Fanuc TP program (LS listing): P004.LS

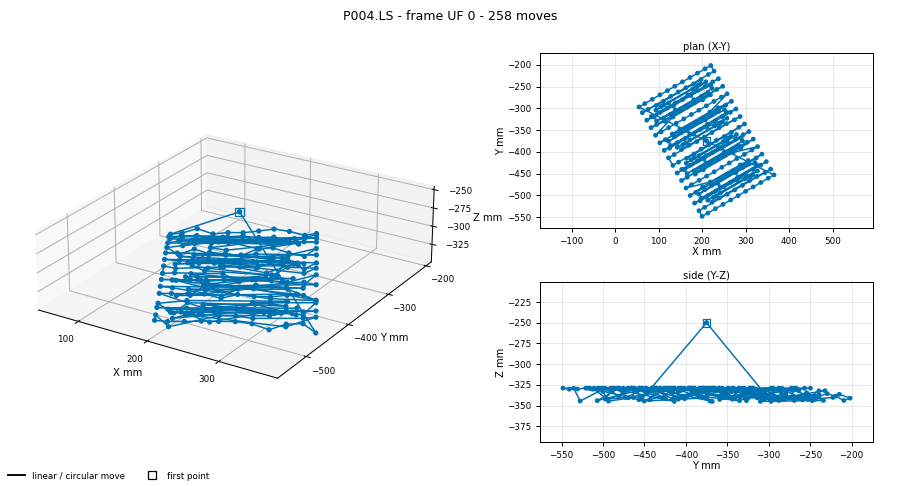
[picture p0: tool path of P004.LS in frame UF 0, 258 of 258 moves have a stored position in this frame; points joined in program order, loops and branches not executed]
/PROG  P004.LS
/ATTR
OWNER       = MNEDITOR;
COMMENT     = "";
PROG_SIZE   = 636;
CREATE      = DATE 23-01-07  TIME 11:59:14;
MODIFIED    = DATE 23-01-07  TIME 12:02:18;
FILE_NAME   = ;
VERSION     = 0;
LINE_COUNT  = 4;
MEMORY_SIZE = 992;
PROTECT     = READ_WRITE;
TCD:  STACK_SIZE	= 0,
      TASK_PRIORITY	= 50,
      TIME_SLICE	= 0,
      BUSY_LAMP_OFF	= 0,
      ABORT_REQUEST	= 0,
      PAUSE_REQUEST	= 0;
DEFAULT_GROUP	= 1,*,*,*,*;
CONTROL_CODE	= 00000000 00000000;
/MN
   1:J P[1] 100% FINE    ;
   2:L P[2] 100mm/sec CNT100    ;
   3:L P[3] 100mm/sec CNT100    ;
   4:L P[4] 100mm/sec CNT100    ;
   5:L P[5] 100mm/sec CNT100    ;
   6:L P[6] 100mm/sec CNT100    ;
   7:L P[7] 100mm/sec CNT100    ;
   8:L P[8] 100mm/sec CNT100    ;
   9:L P[9] 100mm/sec CNT100    ;
   10:L P[10] 100mm/sec CNT100    ;
   11:L P[11] 100mm/sec CNT100    ;
   12:L P[12] 100mm/sec CNT100    ;
   13:L P[13] 100mm/sec CNT100    ;
   14:L P[14] 100mm/sec CNT100    ;
   15:L P[15] 100mm/sec CNT100    ;
   16:L P[16] 100mm/sec CNT100    ;
   17:L P[17] 100mm/sec CNT100    ;
   18:L P[18] 100mm/sec CNT100    ;
   19:L P[19] 100mm/sec CNT100    ;
   20:L P[20] 100mm/sec CNT100    ;
   21:L P[21] 100mm/sec CNT100    ;
   22:L P[22] 100mm/sec CNT100    ;
   23:L P[23] 100mm/sec CNT100    ;
   24:L P[24] 100mm/sec CNT100    ;
   25:L P[25] 100mm/sec CNT100    ;
   26:L P[26] 100mm/sec CNT100    ;
   27:L P[27] 100mm/sec CNT100    ;
   28:L P[28] 100mm/sec CNT100    ;
   29:L P[29] 100mm/sec CNT100    ;
   30:L P[30] 100mm/sec CNT100    ;
   31:L P[31] 100mm/sec CNT100    ;
   32:L P[32] 100mm/sec CNT100    ;
   33:L P[33] 100mm/sec CNT100    ;
   34:L P[34] 100mm/sec CNT100    ;
   35:L P[35] 100mm/sec CNT100    ;
   36:L P[36] 100mm/sec CNT100    ;
   37:L P[37] 100mm/sec CNT100    ;
   38:L P[38] 100mm/sec CNT100    ;
   39:L P[39] 100mm/sec CNT100    ;
   40:L P[40] 100mm/sec CNT100    ;
   41:L P[41] 100mm/sec CNT100    ;
   42:L P[42] 100mm/sec CNT100    ;
   43:L P[43] 100mm/sec CNT100    ;
   44:L P[44] 100mm/sec CNT100    ;
   45:L P[45] 100mm/sec CNT100    ;
   46:L P[46] 100mm/sec CNT100    ;
   47:L P[47] 100mm/sec CNT100    ;
   48:L P[48] 100mm/sec CNT100    ;
   49:L P[49] 100mm/sec CNT100    ;
   50:L P[50] 100mm/sec CNT100    ;
   51:L P[51] 100mm/sec CNT100    ;
   52:L P[52] 100mm/sec CNT100    ;
   53:L P[53] 100mm/sec CNT100    ;
   54:L P[54] 100mm/sec CNT100    ;
   55:L P[55] 100mm/sec CNT100    ;
   56:L P[56] 100mm/sec CNT100    ;
   57:L P[57] 100mm/sec CNT100    ;
   58:L P[58] 100mm/sec CNT100    ;
   59:L P[59] 100mm/sec CNT100    ;
   60:L P[60] 100mm/sec CNT100    ;
   61:L P[61] 100mm/sec CNT100    ;
   62:L P[62] 100mm/sec CNT100    ;
   63:L P[63] 100mm/sec CNT100    ;
   64:L P[64] 100mm/sec CNT100    ;
   65:L P[65] 100mm/sec CNT100    ;
   66:L P[66] 100mm/sec CNT100    ;
   67:L P[67] 100mm/sec CNT100    ;
   68:L P[68] 100mm/sec CNT100    ;
   69:L P[69] 100mm/sec CNT100    ;
   70:L P[70] 100mm/sec CNT100    ;
   71:L P[71] 100mm/sec CNT100    ;
   72:L P[72] 100mm/sec CNT100    ;
   73:L P[73] 100mm/sec CNT100    ;
   74:L P[74] 100mm/sec CNT100    ;
   75:L P[75] 100mm/sec CNT100    ;
   76:L P[76] 100mm/sec CNT100    ;
   77:L P[77] 100mm/sec CNT100    ;
   78:L P[78] 100mm/sec CNT100    ;
   79:L P[79] 100mm/sec CNT100    ;
   80:L P[80] 100mm/sec CNT100    ;
   81:L P[81] 100mm/sec CNT100    ;
   82:L P[82] 100mm/sec CNT100    ;
   83:L P[83] 100mm/sec CNT100    ;
   84:L P[84] 100mm/sec CNT100    ;
   85:L P[85] 100mm/sec CNT100    ;
   86:L P[86] 100mm/sec CNT100    ;
   87:L P[87] 100mm/sec CNT100    ;
   88:L P[88] 100mm/sec CNT100    ;
   89:L P[89] 100mm/sec CNT100    ;
   90:L P[90] 100mm/sec CNT100    ;
   91:L P[91] 100mm/sec CNT100    ;
   92:L P[92] 100mm/sec CNT100    ;
   93:L P[93] 100mm/sec CNT100    ;
   94:L P[94] 100mm/sec CNT100    ;
   95:L P[95] 100mm/sec CNT100    ;
   96:L P[96] 100mm/sec CNT100    ;
   97:L P[97] 100mm/sec CNT100    ;
   98:L P[98] 100mm/sec CNT100    ;
   99:L P[99] 100mm/sec CNT100    ;
   100:L P[100] 100mm/sec CNT100    ;
   101:L P[101] 100mm/sec CNT100    ;
   102:L P[102] 100mm/sec CNT100    ;
   103:L P[103] 100mm/sec CNT100    ;
   104:L P[104] 100mm/sec CNT100    ;
   105:L P[105] 100mm/sec CNT100    ;
   106:L P[106] 100mm/sec CNT100    ;
   107:L P[107] 100mm/sec CNT100    ;
   108:L P[108] 100mm/sec CNT100    ;
   109:L P[109] 100mm/sec CNT100    ;
   110:L P[110] 100mm/sec CNT100    ;
   111:L P[111] 100mm/sec CNT100    ;
   112:L P[112] 100mm/sec CNT100    ;
   113:L P[113] 100mm/sec CNT100    ;
   114:L P[114] 100mm/sec CNT100    ;
   115:L P[115] 100mm/sec CNT100    ;
   116:L P[116] 100mm/sec CNT100    ;
   117:L P[117] 100mm/sec CNT100    ;
   118:L P[118] 100mm/sec CNT100    ;
   119:L P[119] 100mm/sec CNT100    ;
   120:L P[120] 100mm/sec CNT100    ;
   121:L P[121] 100mm/sec CNT100    ;
   122:L P[122] 100mm/sec CNT100    ;
   123:L P[123] 100mm/sec CNT100    ;
   124:L P[124] 100mm/sec CNT100    ;
   125:L P[125] 100mm/sec CNT100    ;
   126:L P[126] 100mm/sec CNT100    ;
   127:L P[127] 100mm/sec CNT100    ;
   128:L P[128] 100mm/sec CNT100    ;
   129:L P[129] 100mm/sec CNT100    ;
   130:L P[130] 100mm/sec CNT100    ;
   131:L P[131] 100mm/sec CNT100    ;
   132:L P[132] 100mm/sec CNT100    ;
   133:L P[133] 100mm/sec CNT100    ;
   134:L P[134] 100mm/sec CNT100    ;
   135:L P[135] 100mm/sec CNT100    ;
   136:L P[136] 100mm/sec CNT100    ;
   137:L P[137] 100mm/sec CNT100    ;
   138:L P[138] 100mm/sec CNT100    ;
   139:L P[139] 100mm/sec CNT100    ;
   140:L P[140] 100mm/sec CNT100    ;
   141:L P[141] 100mm/sec CNT100    ;
   142:L P[142] 100mm/sec CNT100    ;
   143:L P[143] 100mm/sec CNT100    ;
   144:L P[144] 100mm/sec CNT100    ;
   145:L P[145] 100mm/sec CNT100    ;
   146:L P[146] 100mm/sec CNT100    ;
   147:L P[147] 100mm/sec CNT100    ;
   148:L P[148] 100mm/sec CNT100    ;
   149:L P[149] 100mm/sec CNT100    ;
   150:L P[150] 100mm/sec CNT100    ;
   151:L P[151] 100mm/sec CNT100    ;
   152:L P[152] 100mm/sec CNT100    ;
   153:L P[153] 100mm/sec CNT100    ;
   154:L P[154] 100mm/sec CNT100    ;
   155:L P[155] 100mm/sec CNT100    ;
   156:L P[156] 100mm/sec CNT100    ;
   157:L P[157] 100mm/sec CNT100    ;
   158:L P[158] 100mm/sec CNT100    ;
   159:L P[159] 100mm/sec CNT100    ;
   160:L P[160] 100mm/sec CNT100    ;
   161:L P[161] 100mm/sec CNT100    ;
   162:L P[162] 100mm/sec CNT100    ;
   163:L P[163] 100mm/sec CNT100    ;
   164:L P[164] 100mm/sec CNT100    ;
   165:L P[165] 100mm/sec CNT100    ;
   166:L P[166] 100mm/sec CNT100    ;
   167:L P[167] 100mm/sec CNT100    ;
   168:L P[168] 100mm/sec CNT100    ;
   169:L P[169] 100mm/sec CNT100    ;
   170:L P[170] 100mm/sec CNT100    ;
   171:L P[171] 100mm/sec CNT100    ;
   172:L P[172] 100mm/sec CNT100    ;
   173:L P[173] 100mm/sec CNT100    ;
   174:L P[174] 100mm/sec CNT100    ;
   175:L P[175] 100mm/sec CNT100    ;
   176:L P[176] 100mm/sec CNT100    ;
   177:L P[177] 100mm/sec CNT100    ;
   178:L P[178] 100mm/sec CNT100    ;
   179:L P[179] 100mm/sec CNT100    ;
   180:L P[180] 100mm/sec CNT100    ;
   181:L P[181] 100mm/sec CNT100    ;
   182:L P[182] 100mm/sec CNT100    ;
   183:L P[183] 100mm/sec CNT100    ;
   184:L P[184] 100mm/sec CNT100    ;
   185:L P[185] 100mm/sec CNT100    ;
   186:L P[186] 100mm/sec CNT100    ;
   187:L P[187] 100mm/sec CNT100    ;
   188:L P[188] 100mm/sec CNT100    ;
   189:L P[189] 100mm/sec CNT100    ;
   190:L P[190] 100mm/sec CNT100    ;
   191:L P[191] 100mm/sec CNT100    ;
   192:L P[192] 100mm/sec CNT100    ;
   193:L P[193] 100mm/sec CNT100    ;
   194:L P[194] 100mm/sec CNT100    ;
   195:L P[195] 100mm/sec CNT100    ;
   196:L P[196] 100mm/sec CNT100    ;
   197:L P[197] 100mm/sec CNT100    ;
   198:L P[198] 100mm/sec CNT100    ;
   199:L P[199] 100mm/sec CNT100    ;
   200:L P[200] 100mm/sec CNT100    ;
   201:L P[201] 100mm/sec CNT100    ;
   202:L P[202] 100mm/sec CNT100    ;
   203:L P[203] 100mm/sec CNT100    ;
   204:L P[204] 100mm/sec CNT100    ;
   205:L P[205] 100mm/sec CNT100    ;
   206:L P[206] 100mm/sec CNT100    ;
   207:L P[207] 100mm/sec CNT100    ;
   208:L P[208] 100mm/sec CNT100    ;
   209:L P[209] 100mm/sec CNT100    ;
   210:L P[210] 100mm/sec CNT100    ;
   211:L P[211] 100mm/sec CNT100    ;
   212:L P[212] 100mm/sec CNT100    ;
   213:L P[213] 100mm/sec CNT100    ;
   214:L P[214] 100mm/sec CNT100    ;
   215:L P[215] 100mm/sec CNT100    ;
   216:L P[216] 100mm/sec CNT100    ;
   217:L P[217] 100mm/sec CNT100    ;
   218:L P[218] 100mm/sec CNT100    ;
   219:L P[219] 100mm/sec CNT100    ;
   220:L P[220] 100mm/sec CNT100    ;
   221:L P[221] 100mm/sec CNT100    ;
   222:L P[222] 100mm/sec CNT100    ;
   223:L P[223] 100mm/sec CNT100    ;
   224:L P[224] 100mm/sec CNT100    ;
   225:L P[225] 100mm/sec CNT100    ;
   226:L P[226] 100mm/sec CNT100    ;
   227:L P[227] 100mm/sec CNT100    ;
   228:L P[228] 100mm/sec CNT100    ;
   229:L P[229] 100mm/sec CNT100    ;
   230:L P[230] 100mm/sec CNT100    ;
   231:L P[231] 100mm/sec CNT100    ;
   232:L P[232] 100mm/sec CNT100    ;
   233:L P[233] 100mm/sec CNT100    ;
   234:L P[234] 100mm/sec CNT100    ;
   235:L P[235] 100mm/sec CNT100    ;
   236:L P[236] 100mm/sec CNT100    ;
   237:L P[237] 100mm/sec CNT100    ;
   238:L P[238] 100mm/sec CNT100    ;
   239:L P[239] 100mm/sec CNT100    ;
   240:L P[240] 100mm/sec CNT100    ;
   241:L P[241] 100mm/sec CNT100    ;
   242:L P[242] 100mm/sec CNT100    ;
   243:L P[243] 100mm/sec CNT100    ;
   244:L P[244] 100mm/sec CNT100    ;
   245:L P[245] 100mm/sec CNT100    ;
   246:L P[246] 100mm/sec CNT100    ;
   247:L P[247] 100mm/sec CNT100    ;
   248:L P[248] 100mm/sec CNT100    ;
   249:L P[249] 100mm/sec CNT100    ;
   250:L P[250] 100mm/sec CNT100    ;
   251:L P[251] 100mm/sec CNT100    ;
   252:L P[252] 100mm/sec CNT100    ;
   253:L P[253] 100mm/sec CNT100    ;
   254:L P[254] 100mm/sec CNT100    ;
   255:L P[255] 100mm/sec CNT100    ;
   256:L P[256] 100mm/sec CNT100    ;
   257:L P[257] 100mm/sec CNT100    ;
   258:L P[258] 100mm/sec CNT100    ;
/POS
P[1]{
   GP1:
	UF : 0, UT : 6,		CONFIG : 'N U T, 0, 0, 0',
	X =  210.000  mm,	Y =   -375.000  mm,	Z =   -250.000  mm,
	W =  90.000 deg,	P =   0.000 deg,	R =   90.000 deg
};
P[2]{
   GP1:
	UF : 0, UT : 6,		CONFIG : 'N U T, 0, 0, 0',
	X =  54.964  mm,	Y =   -297.033  mm,	Z =   -344.959  mm,
	W =  90.000 deg,	P =   0.000 deg,	R =   90.000 deg
};
P[3]{
   GP1:
	UF : 0, UT : 6,		CONFIG : 'N U T, 0, 0, 0',
	X =  68.285  mm,	Y =   -289.346  mm,	Z =   -342.995  mm,
	W =  90.000 deg,	P =   0.000 deg,	R =   90.000 deg
};
P[4]{
   GP1:
	UF : 0, UT : 6,		CONFIG : 'N U T, 0, 0, 0',
	X =  85.422  mm,	Y =   -279.446  mm,	Z =   -336.480  mm,
	W =  90.000 deg,	P =   0.000 deg,	R =   90.000 deg
};
P[5]{
   GP1:
	UF : 0, UT : 6,		CONFIG : 'N U T, 0, 0, 0',
	X =  102.971  mm,	Y =   -269.165  mm,	Z =   -343.776  mm,
	W =  90.000 deg,	P =   0.000 deg,	R =   90.000 deg
};
P[6]{
   GP1:
	UF : 0, UT : 6,		CONFIG : 'N U T, 0, 0, 0',
	X =  120.213  mm,	Y =   -259.452  mm,	Z =   -341.399  mm,
	W =  90.000 deg,	P =   0.000 deg,	R =   90.000 deg
};
P[7]{
   GP1:
	UF : 0, UT : 6,		CONFIG : 'N U T, 0, 0, 0',
	X =  137.188  mm,	Y =   -249.482  mm,	Z =   -341.375  mm,
	W =  90.000 deg,	P =   0.000 deg,	R =   90.000 deg
};
P[8]{
   GP1:
	UF : 0, UT : 6,		CONFIG : 'N U T, 0, 0, 0',
	X =  154.646  mm,	Y =   -239.297  mm,	Z =   -338.755  mm,
	W =  90.000 deg,	P =   0.000 deg,	R =   90.000 deg
};
P[9]{
   GP1:
	UF : 0, UT : 6,		CONFIG : 'N U T, 0, 0, 0',
	X =  171.892  mm,	Y =   -229.380  mm,	Z =   -335.633  mm,
	W =  90.000 deg,	P =   0.000 deg,	R =   90.000 deg
};
P[10]{
   GP1:
	UF : 0, UT : 6,		CONFIG : 'N U T, 0, 0, 0',
	X =  189.287  mm,	Y =   -219.340  mm,	Z =   -338.627  mm,
	W =  90.000 deg,	P =   0.000 deg,	R =   90.000 deg
};
P[11]{
   GP1:
	UF : 0, UT : 6,		CONFIG : 'N U T, 0, 0, 0',
	X =  206.728  mm,	Y =   -209.278  mm,	Z =   -343.825  mm,
	W =  90.000 deg,	P =   0.000 deg,	R =   90.000 deg
};
P[12]{
   GP1:
	UF : 0, UT : 6,		CONFIG : 'N U T, 0, 0, 0',
	X =  219.749  mm,	Y =   -201.819  mm,	Z =   -341.046  mm,
	W =  90.000 deg,	P =   0.000 deg,	R =   90.000 deg
};
P[13]{
   GP1:
	UF : 0, UT : 6,		CONFIG : 'N U T, 0, 0, 0',
	X =  227.367  mm,	Y =   -214.813  mm,	Z =   -336.366  mm,
	W =  90.000 deg,	P =   0.000 deg,	R =   90.000 deg
};
P[14]{
   GP1:
	UF : 0, UT : 6,		CONFIG : 'N U T, 0, 0, 0',
	X =  214.200  mm,	Y =   -222.393  mm,	Z =   -340.213  mm,
	W =  90.000 deg,	P =   0.000 deg,	R =   90.000 deg
};
P[15]{
   GP1:
	UF : 0, UT : 6,		CONFIG : 'N U T, 0, 0, 0',
	X =  162.666  mm,	Y =   -252.574  mm,	Z =   -342.497  mm,
	W =  90.000 deg,	P =   0.000 deg,	R =   90.000 deg
};
P[16]{
   GP1:
	UF : 0, UT : 6,		CONFIG : 'N U T, 0, 0, 0',
	X =  145.074  mm,	Y =   -262.464  mm,	Z =   -339.220  mm,
	W =  90.000 deg,	P =   0.000 deg,	R =   90.000 deg
};
P[17]{
   GP1:
	UF : 0, UT : 6,		CONFIG : 'N U T, 0, 0, 0',
	X =  127.630  mm,	Y =   -272.610  mm,	Z =   -341.020  mm,
	W =  90.000 deg,	P =   0.000 deg,	R =   90.000 deg
};
P[18]{
   GP1:
	UF : 0, UT : 6,		CONFIG : 'N U T, 0, 0, 0',
	X =  75.778  mm,	Y =   -302.469  mm,	Z =   -340.162  mm,
	W =  90.000 deg,	P =   0.000 deg,	R =   90.000 deg
};
P[19]{
   GP1:
	UF : 0, UT : 6,		CONFIG : 'N U T, 0, 0, 0',
	X =  62.714  mm,	Y =   -310.004  mm,	Z =   -344.947  mm,
	W =  90.000 deg,	P =   0.000 deg,	R =   90.000 deg
};
P[20]{
   GP1:
	UF : 0, UT : 6,		CONFIG : 'N U T, 0, 0, 0',
	X =  197.352  mm,	Y =   -233.917  mm,	Z =   -343.862  mm,
	W =  90.000 deg,	P =   0.000 deg,	R =   90.000 deg
};
P[21]{
   GP1:
	UF : 0, UT : 6,		CONFIG : 'N U T, 0, 0, 0',
	X =  180.545  mm,	Y =   -243.933  mm,	Z =   -339.685  mm,
	W =  90.000 deg,	P =   0.000 deg,	R =   90.000 deg
};
P[22]{
   GP1:
	UF : 0, UT : 6,		CONFIG : 'N U T, 0, 0, 0',
	X =  111.090  mm,	Y =   -283.819  mm,	Z =   -342.744  mm,
	W =  90.000 deg,	P =   0.000 deg,	R =   90.000 deg
};
P[23]{
   GP1:
	UF : 0, UT : 6,		CONFIG : 'N U T, 0, 0, 0',
	X =  94.177  mm,	Y =   -293.763  mm,	Z =   -339.131  mm,
	W =  90.000 deg,	P =   0.000 deg,	R =   90.000 deg
};
P[24]{
   GP1:
	UF : 0, UT : 6,		CONFIG : 'N U T, 0, 0, 0',
	X =  111.350  mm,	Y =   -292.520  mm,	Z =   -339.082  mm,
	W =  90.000 deg,	P =   0.000 deg,	R =   90.000 deg
};
P[25]{
   GP1:
	UF : 0, UT : 6,		CONFIG : 'N U T, 0, 0, 0',
	X =  189.919  mm,	Y =   -247.353  mm,	Z =   -344.029  mm,
	W =  90.000 deg,	P =   0.000 deg,	R =   90.000 deg
};
P[26]{
   GP1:
	UF : 0, UT : 6,		CONFIG : 'N U T, 0, 0, 0',
	X =  195.690  mm,	Y =   -243.952  mm,	Z =   -342.415  mm,
	W =  90.000 deg,	P =   0.000 deg,	R =   90.000 deg
};
P[27]{
   GP1:
	UF : 0, UT : 6,		CONFIG : 'N U T, 0, 0, 0',
	X =  105.186  mm,	Y =   -296.580  mm,	Z =   -339.098  mm,
	W =  90.000 deg,	P =   0.000 deg,	R =   90.000 deg
};
P[28]{
   GP1:
	UF : 0, UT : 6,		CONFIG : 'N U T, 0, 0, 0',
	X =  93.781  mm,	Y =   -304.552  mm,	Z =   -341.716  mm,
	W =  90.000 deg,	P =   0.000 deg,	R =   90.000 deg
};
P[29]{
   GP1:
	UF : 0, UT : 6,		CONFIG : 'N U T, 0, 0, 0',
	X =  122.872  mm,	Y =   -287.580  mm,	Z =   -343.772  mm,
	W =  90.000 deg,	P =   0.000 deg,	R =   90.000 deg
};
P[30]{
   GP1:
	UF : 0, UT : 6,		CONFIG : 'N U T, 0, 0, 0',
	X =  179.007  mm,	Y =   -255.068  mm,	Z =   -339.045  mm,
	W =  90.000 deg,	P =   0.000 deg,	R =   90.000 deg
};
P[31]{
   GP1:
	UF : 0, UT : 6,		CONFIG : 'N U T, 0, 0, 0',
	X =  208.523  mm,	Y =   -239.211  mm,	Z =   -336.820  mm,
	W =  90.000 deg,	P =   0.000 deg,	R =   90.000 deg
};
P[32]{
   GP1:
	UF : 0, UT : 6,		CONFIG : 'N U T, 0, 0, 0',
	X =  167.291  mm,	Y =   -269.037  mm,	Z =   -339.151  mm,
	W =  90.000 deg,	P =   0.000 deg,	R =   90.000 deg
};
P[33]{
   GP1:
	UF : 0, UT : 6,		CONFIG : 'N U T, 0, 0, 0',
	X =  83.192  mm,	Y =   -318.870  mm,	Z =   -338.828  mm,
	W =  90.000 deg,	P =   0.000 deg,	R =   90.000 deg
};
P[34]{
   GP1:
	UF : 0, UT : 6,		CONFIG : 'N U T, 0, 0, 0',
	X =  120.012  mm,	Y =   -299.352  mm,	Z =   -341.751  mm,
	W =  90.000 deg,	P =   0.000 deg,	R =   90.000 deg
};
P[35]{
   GP1:
	UF : 0, UT : 6,		CONFIG : 'N U T, 0, 0, 0',
	X =  138.499  mm,	Y =   -287.571  mm,	Z =   -341.326  mm,
	W =  90.000 deg,	P =   0.000 deg,	R =   90.000 deg
};
P[36]{
   GP1:
	UF : 0, UT : 6,		CONFIG : 'N U T, 0, 0, 0',
	X =  237.306  mm,	Y =   -232.133  mm,	Z =   -332.024  mm,
	W =  90.000 deg,	P =   0.000 deg,	R =   90.000 deg
};
P[37]{
   GP1:
	UF : 0, UT : 6,		CONFIG : 'N U T, 0, 0, 0',
	X =  224.219  mm,	Y =   -239.480  mm,	Z =   -332.129  mm,
	W =  90.000 deg,	P =   0.000 deg,	R =   90.000 deg
};
P[38]{
   GP1:
	UF : 0, UT : 6,		CONFIG : 'N U T, 0, 0, 0',
	X =  206.700  mm,	Y =   -249.866  mm,	Z =   -339.270  mm,
	W =  90.000 deg,	P =   0.000 deg,	R =   90.000 deg
};
P[39]{
   GP1:
	UF : 0, UT : 6,		CONFIG : 'N U T, 0, 0, 0',
	X =  189.366  mm,	Y =   -259.413  mm,	Z =   -342.963  mm,
	W =  90.000 deg,	P =   0.000 deg,	R =   90.000 deg
};
P[40]{
   GP1:
	UF : 0, UT : 6,		CONFIG : 'N U T, 0, 0, 0',
	X =  155.046  mm,	Y =   -279.655  mm,	Z =   -331.747  mm,
	W =  90.000 deg,	P =   0.000 deg,	R =   90.000 deg
};
P[41]{
   GP1:
	UF : 0, UT : 6,		CONFIG : 'N U T, 0, 0, 0',
	X =  103.386  mm,	Y =   -309.449  mm,	Z =   -331.657  mm,
	W =  90.000 deg,	P =   0.000 deg,	R =   90.000 deg
};
P[42]{
   GP1:
	UF : 0, UT : 6,		CONFIG : 'N U T, 0, 0, 0',
	X =  72.723  mm,	Y =   -327.289  mm,	Z =   -333.047  mm,
	W =  90.000 deg,	P =   0.000 deg,	R =   90.000 deg
};
P[43]{
   GP1:
	UF : 0, UT : 6,		CONFIG : 'N U T, 0, 0, 0',
	X =  89.392  mm,	Y =   -320.053  mm,	Z =   -331.771  mm,
	W =  90.000 deg,	P =   0.000 deg,	R =   90.000 deg
};
P[44]{
   GP1:
	UF : 0, UT : 6,		CONFIG : 'N U T, 0, 0, 0',
	X =  134.059  mm,	Y =   -294.533  mm,	Z =   -331.686  mm,
	W =  90.000 deg,	P =   0.000 deg,	R =   90.000 deg
};
P[45]{
   GP1:
	UF : 0, UT : 6,		CONFIG : 'N U T, 0, 0, 0',
	X =  173.844  mm,	Y =   -270.814  mm,	Z =   -331.661  mm,
	W =  90.000 deg,	P =   0.000 deg,	R =   90.000 deg
};
P[46]{
   GP1:
	UF : 0, UT : 6,		CONFIG : 'N U T, 0, 0, 0',
	X =  219.647  mm,	Y =   -247.088  mm,	Z =   -339.207  mm,
	W =  90.000 deg,	P =   0.000 deg,	R =   90.000 deg
};
P[47]{
   GP1:
	UF : 0, UT : 6,		CONFIG : 'N U T, 0, 0, 0',
	X =  222.521  mm,	Y =   -254.254  mm,	Z =   -334.411  mm,
	W =  90.000 deg,	P =   0.000 deg,	R =   90.000 deg
};
P[48]{
   GP1:
	UF : 0, UT : 6,		CONFIG : 'N U T, 0, 0, 0',
	X =  180.771  mm,	Y =   -280.254  mm,	Z =   -342.735  mm,
	W =  90.000 deg,	P =   0.000 deg,	R =   90.000 deg
};
P[49]{
   GP1:
	UF : 0, UT : 6,		CONFIG : 'N U T, 0, 0, 0',
	X =  138.343  mm,	Y =   -304.026  mm,	Z =   -331.765  mm,
	W =  90.000 deg,	P =   0.000 deg,	R =   90.000 deg
};
P[50]{
   GP1:
	UF : 0, UT : 6,		CONFIG : 'N U T, 0, 0, 0',
	X =  95.323  mm,	Y =   -328.988  mm,	Z =   -339.821  mm,
	W =  90.000 deg,	P =   0.000 deg,	R =   90.000 deg
};
P[51]{
   GP1:
	UF : 0, UT : 6,		CONFIG : 'N U T, 0, 0, 0',
	X =  111.227  mm,	Y =   -322.375  mm,	Z =   -329.019  mm,
	W =  90.000 deg,	P =   0.000 deg,	R =   90.000 deg
};
P[52]{
   GP1:
	UF : 0, UT : 6,		CONFIG : 'N U T, 0, 0, 0',
	X =  213.402  mm,	Y =   -263.460  mm,	Z =   -331.340  mm,
	W =  90.000 deg,	P =   0.000 deg,	R =   90.000 deg
};
P[53]{
   GP1:
	UF : 0, UT : 6,		CONFIG : 'N U T, 0, 0, 0',
	X =  198.127  mm,	Y =   -272.813  mm,	Z =   -329.019  mm,
	W =  90.000 deg,	P =   0.000 deg,	R =   90.000 deg
};
P[54]{
   GP1:
	UF : 0, UT : 6,		CONFIG : 'N U T, 0, 0, 0',
	X =  127.780  mm,	Y =   -313.727  mm,	Z =   -340.578  mm,
	W =  90.000 deg,	P =   0.000 deg,	R =   90.000 deg
};
P[55]{
   GP1:
	UF : 0, UT : 6,		CONFIG : 'N U T, 0, 0, 0',
	X =  147.349  mm,	Y =   -306.670  mm,	Z =   -342.340  mm,
	W =  90.000 deg,	P =   0.000 deg,	R =   90.000 deg
};
P[56]{
   GP1:
	UF : 0, UT : 6,		CONFIG : 'N U T, 0, 0, 0',
	X =  233.323  mm,	Y =   -256.738  mm,	Z =   -329.043  mm,
	W =  90.000 deg,	P =   0.000 deg,	R =   90.000 deg
};
P[57]{
   GP1:
	UF : 0, UT : 6,		CONFIG : 'N U T, 0, 0, 0',
	X =  247.216  mm,	Y =   -249.565  mm,	Z =   -329.013  mm,
	W =  90.000 deg,	P =   0.000 deg,	R =   90.000 deg
};
P[58]{
   GP1:
	UF : 0, UT : 6,		CONFIG : 'N U T, 0, 0, 0',
	X =  181.414  mm,	Y =   -287.792  mm,	Z =   -329.000  mm,
	W =  90.000 deg,	P =   0.000 deg,	R =   90.000 deg
};
P[59]{
   GP1:
	UF : 0, UT : 6,		CONFIG : 'N U T, 0, 0, 0',
	X =  165.019  mm,	Y =   -297.017  mm,	Z =   -329.000  mm,
	W =  90.000 deg,	P =   0.000 deg,	R =   90.000 deg
};
P[60]{
   GP1:
	UF : 0, UT : 6,		CONFIG : 'N U T, 0, 0, 0',
	X =  95.378  mm,	Y =   -337.105  mm,	Z =   -330.153  mm,
	W =  90.000 deg,	P =   0.000 deg,	R =   90.000 deg
};
P[61]{
   GP1:
	UF : 0, UT : 6,		CONFIG : 'N U T, 0, 0, 0',
	X =  82.634  mm,	Y =   -344.434  mm,	Z =   -333.012  mm,
	W =  90.000 deg,	P =   0.000 deg,	R =   90.000 deg
};
P[62]{
   GP1:
	UF : 0, UT : 6,		CONFIG : 'N U T, 0, 0, 0',
	X =  114.357  mm,	Y =   -329.935  mm,	Z =   -331.754  mm,
	W =  90.000 deg,	P =   0.000 deg,	R =   90.000 deg
};
P[63]{
   GP1:
	UF : 0, UT : 6,		CONFIG : 'N U T, 0, 0, 0',
	X =  219.042  mm,	Y =   -269.235  mm,	Z =   -329.007  mm,
	W =  90.000 deg,	P =   0.000 deg,	R =   90.000 deg
};
P[64]{
   GP1:
	UF : 0, UT : 6,		CONFIG : 'N U T, 0, 0, 0',
	X =  201.195  mm,	Y =   -280.412  mm,	Z =   -331.367  mm,
	W =  90.000 deg,	P =   0.000 deg,	R =   90.000 deg
};
P[65]{
   GP1:
	UF : 0, UT : 6,		CONFIG : 'N U T, 0, 0, 0',
	X =  132.787  mm,	Y =   -320.108  mm,	Z =   -329.026  mm,
	W =  90.000 deg,	P =   0.000 deg,	R =   90.000 deg
};
P[66]{
   GP1:
	UF : 0, UT : 6,		CONFIG : 'N U T, 0, 0, 0',
	X =  92.843  mm,	Y =   -361.854  mm,	Z =   -330.583  mm,
	W =  90.000 deg,	P =   0.000 deg,	R =   90.000 deg
};
P[67]{
   GP1:
	UF : 0, UT : 6,		CONFIG : 'N U T, 0, 0, 0',
	X =  105.822  mm,	Y =   -354.322  mm,	Z =   -340.290  mm,
	W =  90.000 deg,	P =   0.000 deg,	R =   90.000 deg
};
P[68]{
   GP1:
	UF : 0, UT : 6,		CONFIG : 'N U T, 0, 0, 0',
	X =  123.080  mm,	Y =   -344.334  mm,	Z =   -332.068  mm,
	W =  90.000 deg,	P =   0.000 deg,	R =   90.000 deg
};
P[69]{
   GP1:
	UF : 0, UT : 6,		CONFIG : 'N U T, 0, 0, 0',
	X =  140.433  mm,	Y =   -334.388  mm,	Z =   -338.788  mm,
	W =  90.000 deg,	P =   0.000 deg,	R =   90.000 deg
};
P[70]{
   GP1:
	UF : 0, UT : 6,		CONFIG : 'N U T, 0, 0, 0',
	X =  157.769  mm,	Y =   -324.401  mm,	Z =   -340.163  mm,
	W =  90.000 deg,	P =   0.000 deg,	R =   90.000 deg
};
P[71]{
   GP1:
	UF : 0, UT : 6,		CONFIG : 'N U T, 0, 0, 0',
	X =  175.019  mm,	Y =   -314.311  mm,	Z =   -340.185  mm,
	W =  90.000 deg,	P =   0.000 deg,	R =   90.000 deg
};
P[72]{
   GP1:
	UF : 0, UT : 6,		CONFIG : 'N U T, 0, 0, 0',
	X =  192.396  mm,	Y =   -304.462  mm,	Z =   -330.805  mm,
	W =  90.000 deg,	P =   0.000 deg,	R =   90.000 deg
};
P[73]{
   GP1:
	UF : 0, UT : 6,		CONFIG : 'N U T, 0, 0, 0',
	X =  209.657  mm,	Y =   -294.289  mm,	Z =   -329.043  mm,
	W =  90.000 deg,	P =   0.000 deg,	R =   90.000 deg
};
P[74]{
   GP1:
	UF : 0, UT : 6,		CONFIG : 'N U T, 0, 0, 0',
	X =  227.005  mm,	Y =   -284.264  mm,	Z =   -335.665  mm,
	W =  90.000 deg,	P =   0.000 deg,	R =   90.000 deg
};
P[75]{
   GP1:
	UF : 0, UT : 6,		CONFIG : 'N U T, 0, 0, 0',
	X =  244.227  mm,	Y =   -274.352  mm,	Z =   -340.182  mm,
	W =  90.000 deg,	P =   0.000 deg,	R =   90.000 deg
};
P[76]{
   GP1:
	UF : 0, UT : 6,		CONFIG : 'N U T, 0, 0, 0',
	X =  257.160  mm,	Y =   -266.755  mm,	Z =   -329.000  mm,
	W =  90.000 deg,	P =   0.000 deg,	R =   90.000 deg
};
P[77]{
   GP1:
	UF : 0, UT : 6,		CONFIG : 'N U T, 0, 0, 0',
	X =  217.457  mm,	Y =   -308.775  mm,	Z =   -336.833  mm,
	W =  90.000 deg,	P =   0.000 deg,	R =   90.000 deg
};
P[78]{
   GP1:
	UF : 0, UT : 6,		CONFIG : 'N U T, 0, 0, 0',
	X =  148.690  mm,	Y =   -348.108  mm,	Z =   -329.127  mm,
	W =  90.000 deg,	P =   0.000 deg,	R =   90.000 deg
};
P[79]{
   GP1:
	UF : 0, UT : 6,		CONFIG : 'N U T, 0, 0, 0',
	X =  131.305  mm,	Y =   -359.163  mm,	Z =   -342.666  mm,
	W =  90.000 deg,	P =   0.000 deg,	R =   90.000 deg
};
P[80]{
   GP1:
	UF : 0, UT : 6,		CONFIG : 'N U T, 0, 0, 0',
	X =  236.196  mm,	Y =   -298.720  mm,	Z =   -330.229  mm,
	W =  90.000 deg,	P =   0.000 deg,	R =   90.000 deg
};
P[81]{
   GP1:
	UF : 0, UT : 6,		CONFIG : 'N U T, 0, 0, 0',
	X =  267.157  mm,	Y =   -284.013  mm,	Z =   -329.000  mm,
	W =  90.000 deg,	P =   0.000 deg,	R =   90.000 deg
};
P[82]{
   GP1:
	UF : 0, UT : 6,		CONFIG : 'N U T, 0, 0, 0',
	X =  201.291  mm,	Y =   -321.927  mm,	Z =   -329.001  mm,
	W =  90.000 deg,	P =   0.000 deg,	R =   90.000 deg
};
P[83]{
   GP1:
	UF : 0, UT : 6,		CONFIG : 'N U T, 0, 0, 0',
	X =  185.095  mm,	Y =   -331.576  mm,	Z =   -330.542  mm,
	W =  90.000 deg,	P =   0.000 deg,	R =   90.000 deg
};
P[84]{
   GP1:
	UF : 0, UT : 6,		CONFIG : 'N U T, 0, 0, 0',
	X =  115.534  mm,	Y =   -372.015  mm,	Z =   -329.000  mm,
	W =  90.000 deg,	P =   0.000 deg,	R =   90.000 deg
};
P[85]{
   GP1:
	UF : 0, UT : 6,		CONFIG : 'N U T, 0, 0, 0',
	X =  102.734  mm,	Y =   -379.332  mm,	Z =   -329.028  mm,
	W =  90.000 deg,	P =   0.000 deg,	R =   90.000 deg
};
P[86]{
   GP1:
	UF : 0, UT : 6,		CONFIG : 'N U T, 0, 0, 0',
	X =  167.910  mm,	Y =   -342.172  mm,	Z =   -329.000  mm,
	W =  90.000 deg,	P =   0.000 deg,	R =   90.000 deg
};
P[87]{
   GP1:
	UF : 0, UT : 6,		CONFIG : 'N U T, 0, 0, 0',
	X =  254.271  mm,	Y =   -292.688  mm,	Z =   -341.050  mm,
	W =  90.000 deg,	P =   0.000 deg,	R =   90.000 deg
};
P[88]{
   GP1:
	UF : 0, UT : 6,		CONFIG : 'N U T, 0, 0, 0',
	X =  222.397  mm,	Y =   -315.138  mm,	Z =   -330.212  mm,
	W =  90.000 deg,	P =   0.000 deg,	R =   90.000 deg
};
P[89]{
   GP1:
	UF : 0, UT : 6,		CONFIG : 'N U T, 0, 0, 0',
	X =  151.725  mm,	Y =   -355.659  mm,	Z =   -329.013  mm,
	W =  90.000 deg,	P =   0.000 deg,	R =   90.000 deg
};
P[90]{
   GP1:
	UF : 0, UT : 6,		CONFIG : 'N U T, 0, 0, 0',
	X =  136.256  mm,	Y =   -365.631  mm,	Z =   -329.000  mm,
	W =  90.000 deg,	P =   0.000 deg,	R =   90.000 deg
};
P[91]{
   GP1:
	UF : 0, UT : 6,		CONFIG : 'N U T, 0, 0, 0',
	X =  238.230  mm,	Y =   -306.479  mm,	Z =   -331.261  mm,
	W =  90.000 deg,	P =   0.000 deg,	R =   90.000 deg
};
P[92]{
   GP1:
	UF : 0, UT : 6,		CONFIG : 'N U T, 0, 0, 0',
	X =  207.228  mm,	Y =   -326.792  mm,	Z =   -344.003  mm,
	W =  90.000 deg,	P =   0.000 deg,	R =   90.000 deg
};
P[93]{
   GP1:
	UF : 0, UT : 6,		CONFIG : 'N U T, 0, 0, 0',
	X =  165.371  mm,	Y =   -351.259  mm,	Z =   -335.727  mm,
	W =  90.000 deg,	P =   0.000 deg,	R =   90.000 deg
};
P[94]{
   GP1:
	UF : 0, UT : 6,		CONFIG : 'N U T, 0, 0, 0',
	X =  122.935  mm,	Y =   -375.735  mm,	Z =   -330.203  mm,
	W =  90.000 deg,	P =   0.000 deg,	R =   90.000 deg
};
P[95]{
   GP1:
	UF : 0, UT : 6,		CONFIG : 'N U T, 0, 0, 0',
	X =  251.034  mm,	Y =   -303.404  mm,	Z =   -336.716  mm,
	W =  90.000 deg,	P =   0.000 deg,	R =   90.000 deg
};
P[96]{
   GP1:
	UF : 0, UT : 6,		CONFIG : 'N U T, 0, 0, 0',
	X =  255.794  mm,	Y =   -309.411  mm,	Z =   -336.576  mm,
	W =  90.000 deg,	P =   0.000 deg,	R =   90.000 deg
};
P[97]{
   GP1:
	UF : 0, UT : 6,		CONFIG : 'N U T, 0, 0, 0',
	X =  171.631  mm,	Y =   -359.385  mm,	Z =   -339.120  mm,
	W =  90.000 deg,	P =   0.000 deg,	R =   90.000 deg
};
P[98]{
   GP1:
	UF : 0, UT : 6,		CONFIG : 'N U T, 0, 0, 0',
	X =  211.999  mm,	Y =   -337.291  mm,	Z =   -331.382  mm,
	W =  90.000 deg,	P =   0.000 deg,	R =   90.000 deg
};
P[99]{
   GP1:
	UF : 0, UT : 6,		CONFIG : 'N U T, 0, 0, 0',
	X =  127.390  mm,	Y =   -385.610  mm,	Z =   -331.661  mm,
	W =  90.000 deg,	P =   0.000 deg,	R =   90.000 deg
};
P[100]{
   GP1:
	UF : 0, UT : 6,		CONFIG : 'N U T, 0, 0, 0',
	X =  112.767  mm,	Y =   -396.676  mm,	Z =   -329.000  mm,
	W =  90.000 deg,	P =   0.000 deg,	R =   90.000 deg
};
P[101]{
   GP1:
	UF : 0, UT : 6,		CONFIG : 'N U T, 0, 0, 0',
	X =  143.369  mm,	Y =   -379.012  mm,	Z =   -329.000  mm,
	W =  90.000 deg,	P =   0.000 deg,	R =   90.000 deg
};
P[102]{
   GP1:
	UF : 0, UT : 6,		CONFIG : 'N U T, 0, 0, 0',
	X =  160.556  mm,	Y =   -369.393  mm,	Z =   -329.029  mm,
	W =  90.000 deg,	P =   0.000 deg,	R =   90.000 deg
};
P[103]{
   GP1:
	UF : 0, UT : 6,		CONFIG : 'N U T, 0, 0, 0',
	X =  194.810  mm,	Y =   -349.163  mm,	Z =   -329.000  mm,
	W =  90.000 deg,	P =   0.000 deg,	R =   90.000 deg
};
P[104]{
   GP1:
	UF : 0, UT : 6,		CONFIG : 'N U T, 0, 0, 0',
	X =  246.781  mm,	Y =   -319.004  mm,	Z =   -329.000  mm,
	W =  90.000 deg,	P =   0.000 deg,	R =   90.000 deg
};
P[105]{
   GP1:
	UF : 0, UT : 6,		CONFIG : 'N U T, 0, 0, 0',
	X =  264.592  mm,	Y =   -309.341  mm,	Z =   -339.203  mm,
	W =  90.000 deg,	P =   0.000 deg,	R =   90.000 deg
};
P[106]{
   GP1:
	UF : 0, UT : 6,		CONFIG : 'N U T, 0, 0, 0',
	X =  277.449  mm,	Y =   -301.566  mm,	Z =   -330.833  mm,
	W =  90.000 deg,	P =   0.000 deg,	R =   90.000 deg
};
P[107]{
   GP1:
	UF : 0, UT : 6,		CONFIG : 'N U T, 0, 0, 0',
	X =  230.019  mm,	Y =   -329.393  mm,	Z =   -329.028  mm,
	W =  90.000 deg,	P =   0.000 deg,	R =   90.000 deg
};
P[108]{
   GP1:
	UF : 0, UT : 6,		CONFIG : 'N U T, 0, 0, 0',
	X =  125.050  mm,	Y =   -391.579  mm,	Z =   -334.380  mm,
	W =  90.000 deg,	P =   0.000 deg,	R =   90.000 deg
};
P[109]{
   GP1:
	UF : 0, UT : 6,		CONFIG : 'N U T, 0, 0, 0',
	X =  179.919  mm,	Y =   -359.513  mm,	Z =   -329.008  mm,
	W =  90.000 deg,	P =   0.000 deg,	R =   90.000 deg
};
P[110]{
   GP1:
	UF : 0, UT : 6,		CONFIG : 'N U T, 0, 0, 0',
	X =  210.213  mm,	Y =   -343.666  mm,	Z =   -329.000  mm,
	W =  90.000 deg,	P =   0.000 deg,	R =   90.000 deg
};
P[111]{
   GP1:
	UF : 0, UT : 6,		CONFIG : 'N U T, 0, 0, 0',
	X =  256.759  mm,	Y =   -323.038  mm,	Z =   -329.000  mm,
	W =  90.000 deg,	P =   0.000 deg,	R =   90.000 deg
};
P[112]{
   GP1:
	UF : 0, UT : 6,		CONFIG : 'N U T, 0, 0, 0',
	X =  228.321  mm,	Y =   -340.634  mm,	Z =   -341.366  mm,
	W =  90.000 deg,	P =   0.000 deg,	R =   90.000 deg
};
P[113]{
   GP1:
	UF : 0, UT : 6,		CONFIG : 'N U T, 0, 0, 0',
	X =  171.874  mm,	Y =   -373.116  mm,	Z =   -329.042  mm,
	W =  90.000 deg,	P =   0.000 deg,	R =   90.000 deg
};
P[114]{
   GP1:
	UF : 0, UT : 6,		CONFIG : 'N U T, 0, 0, 0',
	X =  142.948  mm,	Y =   -389.644  mm,	Z =   -329.002  mm,
	W =  90.000 deg,	P =   0.000 deg,	R =   90.000 deg
};
P[115]{
   GP1:
	UF : 0, UT : 6,		CONFIG : 'N U T, 0, 0, 0',
	X =  155.686  mm,	Y =   -383.722  mm,	Z =   -329.013  mm,
	W =  90.000 deg,	P =   0.000 deg,	R =   90.000 deg
};
P[116]{
   GP1:
	UF : 0, UT : 6,		CONFIG : 'N U T, 0, 0, 0',
	X =  246.698  mm,	Y =   -331.373  mm,	Z =   -329.036  mm,
	W =  90.000 deg,	P =   0.000 deg,	R =   90.000 deg
};
P[117]{
   GP1:
	UF : 0, UT : 6,		CONFIG : 'N U T, 0, 0, 0',
	X =  240.343  mm,	Y =   -335.183  mm,	Z =   -344.054  mm,
	W =  90.000 deg,	P =   0.000 deg,	R =   90.000 deg
};
P[118]{
   GP1:
	UF : 0, UT : 6,		CONFIG : 'N U T, 0, 0, 0',
	X =  162.006  mm,	Y =   -380.425  mm,	Z =   -339.105  mm,
	W =  90.000 deg,	P =   0.000 deg,	R =   90.000 deg
};
P[119]{
   GP1:
	UF : 0, UT : 6,		CONFIG : 'N U T, 0, 0, 0',
	X =  152.570  mm,	Y =   -394.661  mm,	Z =   -329.000  mm,
	W =  90.000 deg,	P =   0.000 deg,	R =   90.000 deg
};
P[120]{
   GP1:
	UF : 0, UT : 6,		CONFIG : 'N U T, 0, 0, 0',
	X =  169.614  mm,	Y =   -384.897  mm,	Z =   -331.867  mm,
	W =  90.000 deg,	P =   0.000 deg,	R =   90.000 deg
};
P[121]{
   GP1:
	UF : 0, UT : 6,		CONFIG : 'N U T, 0, 0, 0',
	X =  238.902  mm,	Y =   -344.786  mm,	Z =   -340.586  mm,
	W =  90.000 deg,	P =   0.000 deg,	R =   90.000 deg
};
P[122]{
   GP1:
	UF : 0, UT : 6,		CONFIG : 'N U T, 0, 0, 0',
	X =  255.708  mm,	Y =   -335.320  mm,	Z =   -329.019  mm,
	W =  90.000 deg,	P =   0.000 deg,	R =   90.000 deg
};
P[123]{
   GP1:
	UF : 0, UT : 6,		CONFIG : 'N U T, 0, 0, 0',
	X =  287.230  mm,	Y =   -318.953  mm,	Z =   -329.000  mm,
	W =  90.000 deg,	P =   0.000 deg,	R =   90.000 deg
};
P[124]{
   GP1:
	UF : 0, UT : 6,		CONFIG : 'N U T, 0, 0, 0',
	X =  274.144  mm,	Y =   -326.412  mm,	Z =   -336.348  mm,
	W =  90.000 deg,	P =   0.000 deg,	R =   90.000 deg
};
P[125]{
   GP1:
	UF : 0, UT : 6,		CONFIG : 'N U T, 0, 0, 0',
	X =  222.566  mm,	Y =   -355.680  mm,	Z =   -330.140  mm,
	W =  90.000 deg,	P =   0.000 deg,	R =   90.000 deg
};
P[126]{
   GP1:
	UF : 0, UT : 6,		CONFIG : 'N U T, 0, 0, 0',
	X =  205.127  mm,	Y =   -366.356  mm,	Z =   -329.002  mm,
	W =  90.000 deg,	P =   0.000 deg,	R =   90.000 deg
};
P[127]{
   GP1:
	UF : 0, UT : 6,		CONFIG : 'N U T, 0, 0, 0',
	X =  187.649  mm,	Y =   -376.444  mm,	Z =   -329.038  mm,
	W =  90.000 deg,	P =   0.000 deg,	R =   90.000 deg
};
P[128]{
   GP1:
	UF : 0, UT : 6,		CONFIG : 'N U T, 0, 0, 0',
	X =  135.693  mm,	Y =   -406.364  mm,	Z =   -332.079  mm,
	W =  90.000 deg,	P =   0.000 deg,	R =   90.000 deg
};
P[129]{
   GP1:
	UF : 0, UT : 6,		CONFIG : 'N U T, 0, 0, 0',
	X =  122.715  mm,	Y =   -413.804  mm,	Z =   -329.001  mm,
	W =  90.000 deg,	P =   0.000 deg,	R =   90.000 deg
};
P[130]{
   GP1:
	UF : 0, UT : 6,		CONFIG : 'N U T, 0, 0, 0',
	X =  132.757  mm,	Y =   -431.210  mm,	Z =   -329.959  mm,
	W =  90.000 deg,	P =   0.000 deg,	R =   90.000 deg
};
P[131]{
   GP1:
	UF : 0, UT : 6,		CONFIG : 'N U T, 0, 0, 0',
	X =  145.670  mm,	Y =   -423.684  mm,	Z =   -329.000  mm,
	W =  90.000 deg,	P =   0.000 deg,	R =   90.000 deg
};
P[132]{
   GP1:
	UF : 0, UT : 6,		CONFIG : 'N U T, 0, 0, 0',
	X =  197.579  mm,	Y =   -393.900  mm,	Z =   -329.018  mm,
	W =  90.000 deg,	P =   0.000 deg,	R =   90.000 deg
};
P[133]{
   GP1:
	UF : 0, UT : 6,		CONFIG : 'N U T, 0, 0, 0',
	X =  214.967  mm,	Y =   -383.755  mm,	Z =   -339.766  mm,
	W =  90.000 deg,	P =   0.000 deg,	R =   90.000 deg
};
P[134]{
   GP1:
	UF : 0, UT : 6,		CONFIG : 'N U T, 0, 0, 0',
	X =  232.673  mm,	Y =   -373.776  mm,	Z =   -336.847  mm,
	W =  90.000 deg,	P =   0.000 deg,	R =   90.000 deg
};
P[135]{
   GP1:
	UF : 0, UT : 6,		CONFIG : 'N U T, 0, 0, 0',
	X =  284.419  mm,	Y =   -343.550  mm,	Z =   -342.364  mm,
	W =  90.000 deg,	P =   0.000 deg,	R =   90.000 deg
};
P[136]{
   GP1:
	UF : 0, UT : 6,		CONFIG : 'N U T, 0, 0, 0',
	X =  297.248  mm,	Y =   -336.060  mm,	Z =   -329.024  mm,
	W =  90.000 deg,	P =   0.000 deg,	R =   90.000 deg
};
P[137]{
   GP1:
	UF : 0, UT : 6,		CONFIG : 'N U T, 0, 0, 0',
	X =  267.211  mm,	Y =   -355.124  mm,	Z =   -338.981  mm,
	W =  90.000 deg,	P =   0.000 deg,	R =   90.000 deg
};
P[138]{
   GP1:
	UF : 0, UT : 6,		CONFIG : 'N U T, 0, 0, 0',
	X =  164.270  mm,	Y =   -414.926  mm,	Z =   -329.021  mm,
	W =  90.000 deg,	P =   0.000 deg,	R =   90.000 deg
};
P[139]{
   GP1:
	UF : 0, UT : 6,		CONFIG : 'N U T, 0, 0, 0',
	X =  181.158  mm,	Y =   -405.144  mm,	Z =   -339.099  mm,
	W =  90.000 deg,	P =   0.000 deg,	R =   90.000 deg
};
P[140]{
   GP1:
	UF : 0, UT : 6,		CONFIG : 'N U T, 0, 0, 0',
	X =  250.625  mm,	Y =   -365.135  mm,	Z =   -329.123  mm,
	W =  90.000 deg,	P =   0.000 deg,	R =   90.000 deg
};
P[141]{
   GP1:
	UF : 0, UT : 6,		CONFIG : 'N U T, 0, 0, 0',
	X =  266.312  mm,	Y =   -364.946  mm,	Z =   -332.108  mm,
	W =  90.000 deg,	P =   0.000 deg,	R =   90.000 deg
};
P[142]{
   GP1:
	UF : 0, UT : 6,		CONFIG : 'N U T, 0, 0, 0',
	X =  260.098  mm,	Y =   -368.362  mm,	Z =   -329.014  mm,
	W =  90.000 deg,	P =   0.000 deg,	R =   90.000 deg
};
P[143]{
   GP1:
	UF : 0, UT : 6,		CONFIG : 'N U T, 0, 0, 0',
	X =  181.653  mm,	Y =   -413.645  mm,	Z =   -339.826  mm,
	W =  90.000 deg,	P =   0.000 deg,	R =   90.000 deg
};
P[144]{
   GP1:
	UF : 0, UT : 6,		CONFIG : 'N U T, 0, 0, 0',
	X =  174.967  mm,	Y =   -417.987  mm,	Z =   -329.000  mm,
	W =  90.000 deg,	P =   0.000 deg,	R =   90.000 deg
};
P[145]{
   GP1:
	UF : 0, UT : 6,		CONFIG : 'N U T, 0, 0, 0',
	X =  248.912  mm,	Y =   -376.390  mm,	Z =   -329.117  mm,
	W =  90.000 deg,	P =   0.000 deg,	R =   90.000 deg
};
P[146]{
   GP1:
	UF : 0, UT : 6,		CONFIG : 'N U T, 0, 0, 0',
	X =  192.836  mm,	Y =   -408.880  mm,	Z =   -342.211  mm,
	W =  90.000 deg,	P =   0.000 deg,	R =   90.000 deg
};
P[147]{
   GP1:
	UF : 0, UT : 6,		CONFIG : 'N U T, 0, 0, 0',
	X =  163.435  mm,	Y =   -426.067  mm,	Z =   -329.045  mm,
	W =  90.000 deg,	P =   0.000 deg,	R =   90.000 deg
};
P[148]{
   GP1:
	UF : 0, UT : 6,		CONFIG : 'N U T, 0, 0, 0',
	X =  278.644  mm,	Y =   -360.412  mm,	Z =   -329.000  mm,
	W =  90.000 deg,	P =   0.000 deg,	R =   90.000 deg
};
P[149]{
   GP1:
	UF : 0, UT : 6,		CONFIG : 'N U T, 0, 0, 0',
	X =  237.200  mm,	Y =   -390.225  mm,	Z =   -329.043  mm,
	W =  90.000 deg,	P =   0.000 deg,	R =   90.000 deg
};
P[150]{
   GP1:
	UF : 0, UT : 6,		CONFIG : 'N U T, 0, 0, 0',
	X =  153.129  mm,	Y =   -440.137  mm,	Z =   -330.554  mm,
	W =  90.000 deg,	P =   0.000 deg,	R =   90.000 deg
};
P[151]{
   GP1:
	UF : 0, UT : 6,		CONFIG : 'N U T, 0, 0, 0',
	X =  259.444  mm,	Y =   -380.403  mm,	Z =   -329.000  mm,
	W =  90.000 deg,	P =   0.000 deg,	R =   90.000 deg
};
P[152]{
   GP1:
	UF : 0, UT : 6,		CONFIG : 'N U T, 0, 0, 0',
	X =  208.491  mm,	Y =   -408.857  mm,	Z =   -329.013  mm,
	W =  90.000 deg,	P =   0.000 deg,	R =   90.000 deg
};
P[153]{
   GP1:
	UF : 0, UT : 6,		CONFIG : 'N U T, 0, 0, 0',
	X =  190.036  mm,	Y =   -420.531  mm,	Z =   -329.068  mm,
	W =  90.000 deg,	P =   0.000 deg,	R =   90.000 deg
};
P[154]{
   GP1:
	UF : 0, UT : 6,		CONFIG : 'N U T, 0, 0, 0',
	X =  142.640  mm,	Y =   -448.526  mm,	Z =   -329.028  mm,
	W =  90.000 deg,	P =   0.000 deg,	R =   90.000 deg
};
P[155]{
   GP1:
	UF : 0, UT : 6,		CONFIG : 'N U T, 0, 0, 0',
	X =  173.073  mm,	Y =   -430.710  mm,	Z =   -329.000  mm,
	W =  90.000 deg,	P =   0.000 deg,	R =   90.000 deg
};
P[156]{
   GP1:
	UF : 0, UT : 6,		CONFIG : 'N U T, 0, 0, 0',
	X =  225.006  mm,	Y =   -400.988  mm,	Z =   -339.076  mm,
	W =  90.000 deg,	P =   0.000 deg,	R =   90.000 deg
};
P[157]{
   GP1:
	UF : 0, UT : 6,		CONFIG : 'N U T, 0, 0, 0',
	X =  276.692  mm,	Y =   -371.053  mm,	Z =   -331.312  mm,
	W =  90.000 deg,	P =   0.000 deg,	R =   90.000 deg
};
P[158]{
   GP1:
	UF : 0, UT : 6,		CONFIG : 'N U T, 0, 0, 0',
	X =  294.162  mm,	Y =   -360.651  mm,	Z =   -330.009  mm,
	W =  90.000 deg,	P =   0.000 deg,	R =   90.000 deg
};
P[159]{
   GP1:
	UF : 0, UT : 6,		CONFIG : 'N U T, 0, 0, 0',
	X =  307.317  mm,	Y =   -353.442  mm,	Z =   -333.010  mm,
	W =  90.000 deg,	P =   0.000 deg,	R =   90.000 deg
};
P[160]{
   GP1:
	UF : 0, UT : 6,		CONFIG : 'N U T, 0, 0, 0',
	X =  243.794  mm,	Y =   -392.133  mm,	Z =   -334.255  mm,
	W =  90.000 deg,	P =   0.000 deg,	R =   90.000 deg
};
P[161]{
   GP1:
	UF : 0, UT : 6,		CONFIG : 'N U T, 0, 0, 0',
	X =  204.143  mm,	Y =   -415.878  mm,	Z =   -342.175  mm,
	W =  90.000 deg,	P =   0.000 deg,	R =   90.000 deg
};
P[162]{
   GP1:
	UF : 0, UT : 6,		CONFIG : 'N U T, 0, 0, 0',
	X =  159.508  mm,	Y =   -441.410  mm,	Z =   -329.002  mm,
	W =  90.000 deg,	P =   0.000 deg,	R =   90.000 deg
};
P[163]{
   GP1:
	UF : 0, UT : 6,		CONFIG : 'N U T, 0, 0, 0',
	X =  289.542  mm,	Y =   -368.075  mm,	Z =   -344.978  mm,
	W =  90.000 deg,	P =   0.000 deg,	R =   90.000 deg
};
P[164]{
   GP1:
	UF : 0, UT : 6,		CONFIG : 'N U T, 0, 0, 0',
	X =  292.474  mm,	Y =   -375.225  mm,	Z =   -340.604  mm,
	W =  90.000 deg,	P =   0.000 deg,	R =   90.000 deg
};
P[165]{
   GP1:
	UF : 0, UT : 6,		CONFIG : 'N U T, 0, 0, 0',
	X =  165.534  mm,	Y =   -450.086  mm,	Z =   -344.550  mm,
	W =  90.000 deg,	P =   0.000 deg,	R =   90.000 deg
};
P[166]{
   GP1:
	UF : 0, UT : 6,		CONFIG : 'N U T, 0, 0, 0',
	X =  208.283  mm,	Y =   -425.551  mm,	Z =   -330.485  mm,
	W =  90.000 deg,	P =   0.000 deg,	R =   90.000 deg
};
P[167]{
   GP1:
	UF : 0, UT : 6,		CONFIG : 'N U T, 0, 0, 0',
	X =  250.616  mm,	Y =   -401.489  mm,	Z =   -329.000  mm,
	W =  90.000 deg,	P =   0.000 deg,	R =   90.000 deg
};
P[168]{
   GP1:
	UF : 0, UT : 6,		CONFIG : 'N U T, 0, 0, 0',
	X =  283.660  mm,	Y =   -384.605  mm,	Z =   -330.604  mm,
	W =  90.000 deg,	P =   0.000 deg,	R =   90.000 deg
};
P[169]{
   GP1:
	UF : 0, UT : 6,		CONFIG : 'N U T, 0, 0, 0',
	X =  267.974  mm,	Y =   -394.062  mm,	Z =   -329.000  mm,
	W =  90.000 deg,	P =   0.000 deg,	R =   90.000 deg
};
P[170]{
   GP1:
	UF : 0, UT : 6,		CONFIG : 'N U T, 0, 0, 0',
	X =  181.438  mm,	Y =   -443.460  mm,	Z =   -342.947  mm,
	W =  90.000 deg,	P =   0.000 deg,	R =   90.000 deg
};
P[171]{
   GP1:
	UF : 0, UT : 6,		CONFIG : 'N U T, 0, 0, 0',
	X =  197.787  mm,	Y =   -434.916  mm,	Z =   -329.022  mm,
	W =  90.000 deg,	P =   0.000 deg,	R =   90.000 deg
};
P[172]{
   GP1:
	UF : 0, UT : 6,		CONFIG : 'N U T, 0, 0, 0',
	X =  303.234  mm,	Y =   -378.012  mm,	Z =   -329.000  mm,
	W =  90.000 deg,	P =   0.000 deg,	R =   90.000 deg
};
P[173]{
   GP1:
	UF : 0, UT : 6,		CONFIG : 'N U T, 0, 0, 0',
	X =  152.681  mm,	Y =   -465.814  mm,	Z =   -329.000  mm,
	W =  90.000 deg,	P =   0.000 deg,	R =   90.000 deg
};
P[174]{
   GP1:
	UF : 0, UT : 6,		CONFIG : 'N U T, 0, 0, 0',
	X =  165.397  mm,	Y =   -458.286  mm,	Z =   -330.814  mm,
	W =  90.000 deg,	P =   0.000 deg,	R =   90.000 deg
};
P[175]{
   GP1:
	UF : 0, UT : 6,		CONFIG : 'N U T, 0, 0, 0',
	X =  217.411  mm,	Y =   -428.002  mm,	Z =   -340.963  mm,
	W =  90.000 deg,	P =   0.000 deg,	R =   90.000 deg
};
P[176]{
   GP1:
	UF : 0, UT : 6,		CONFIG : 'N U T, 0, 0, 0',
	X =  234.903  mm,	Y =   -418.324  mm,	Z =   -331.234  mm,
	W =  90.000 deg,	P =   0.000 deg,	R =   90.000 deg
};
P[177]{
   GP1:
	UF : 0, UT : 6,		CONFIG : 'N U T, 0, 0, 0',
	X =  251.379  mm,	Y =   -409.077  mm,	Z =   -330.456  mm,
	W =  90.000 deg,	P =   0.000 deg,	R =   90.000 deg
};
P[178]{
   GP1:
	UF : 0, UT : 6,		CONFIG : 'N U T, 0, 0, 0',
	X =  317.343  mm,	Y =   -370.943  mm,	Z =   -344.537  mm,
	W =  90.000 deg,	P =   0.000 deg,	R =   90.000 deg
};
P[179]{
   GP1:
	UF : 0, UT : 6,		CONFIG : 'N U T, 0, 0, 0',
	X =  288.975  mm,	Y =   -390.612  mm,	Z =   -329.003  mm,
	W =  90.000 deg,	P =   0.000 deg,	R =   90.000 deg
};
P[180]{
   GP1:
	UF : 0, UT : 6,		CONFIG : 'N U T, 0, 0, 0',
	X =  184.192  mm,	Y =   -451.263  mm,	Z =   -330.829  mm,
	W =  90.000 deg,	P =   0.000 deg,	R =   90.000 deg
};
P[181]{
   GP1:
	UF : 0, UT : 6,		CONFIG : 'N U T, 0, 0, 0',
	X =  202.628  mm,	Y =   -441.462  mm,	Z =   -331.710  mm,
	W =  90.000 deg,	P =   0.000 deg,	R =   90.000 deg
};
P[182]{
   GP1:
	UF : 0, UT : 6,		CONFIG : 'N U T, 0, 0, 0',
	X =  271.029  mm,	Y =   -401.573  mm,	Z =   -341.750  mm,
	W =  90.000 deg,	P =   0.000 deg,	R =   90.000 deg
};
P[183]{
   GP1:
	UF : 0, UT : 6,		CONFIG : 'N U T, 0, 0, 0',
	X =  327.284  mm,	Y =   -388.067  mm,	Z =   -335.667  mm,
	W =  90.000 deg,	P =   0.000 deg,	R =   90.000 deg
};
P[184]{
   GP1:
	UF : 0, UT : 6,		CONFIG : 'N U T, 0, 0, 0',
	X =  314.252  mm,	Y =   -395.590  mm,	Z =   -329.022  mm,
	W =  90.000 deg,	P =   0.000 deg,	R =   90.000 deg
};
P[185]{
   GP1:
	UF : 0, UT : 6,		CONFIG : 'N U T, 0, 0, 0',
	X =  297.107  mm,	Y =   -405.873  mm,	Z =   -329.043  mm,
	W =  90.000 deg,	P =   0.000 deg,	R =   90.000 deg
};
P[186]{
   GP1:
	UF : 0, UT : 6,		CONFIG : 'N U T, 0, 0, 0',
	X =  279.649  mm,	Y =   -415.607  mm,	Z =   -331.541  mm,
	W =  90.000 deg,	P =   0.000 deg,	R =   90.000 deg
};
P[187]{
   GP1:
	UF : 0, UT : 6,		CONFIG : 'N U T, 0, 0, 0',
	X =  262.322  mm,	Y =   -425.645  mm,	Z =   -331.310  mm,
	W =  90.000 deg,	P =   0.000 deg,	R =   90.000 deg
};
P[188]{
   GP1:
	UF : 0, UT : 6,		CONFIG : 'N U T, 0, 0, 0',
	X =  245.104  mm,	Y =   -435.630  mm,	Z =   -329.029  mm,
	W =  90.000 deg,	P =   0.000 deg,	R =   90.000 deg
};
P[189]{
   GP1:
	UF : 0, UT : 6,		CONFIG : 'N U T, 0, 0, 0',
	X =  227.702  mm,	Y =   -445.858  mm,	Z =   -334.320  mm,
	W =  90.000 deg,	P =   0.000 deg,	R =   90.000 deg
};
P[190]{
   GP1:
	UF : 0, UT : 6,		CONFIG : 'N U T, 0, 0, 0',
	X =  210.397  mm,	Y =   -455.681  mm,	Z =   -329.000  mm,
	W =  90.000 deg,	P =   0.000 deg,	R =   90.000 deg
};
P[191]{
   GP1:
	UF : 0, UT : 6,		CONFIG : 'N U T, 0, 0, 0',
	X =  193.126  mm,	Y =   -465.589  mm,	Z =   -329.041  mm,
	W =  90.000 deg,	P =   0.000 deg,	R =   90.000 deg
};
P[192]{
   GP1:
	UF : 0, UT : 6,		CONFIG : 'N U T, 0, 0, 0',
	X =  175.448  mm,	Y =   -475.616  mm,	Z =   -329.022  mm,
	W =  90.000 deg,	P =   0.000 deg,	R =   90.000 deg
};
P[193]{
   GP1:
	UF : 0, UT : 6,		CONFIG : 'N U T, 0, 0, 0',
	X =  162.767  mm,	Y =   -483.187  mm,	Z =   -329.035  mm,
	W =  90.000 deg,	P =   0.000 deg,	R =   90.000 deg
};
P[194]{
   GP1:
	UF : 0, UT : 6,		CONFIG : 'N U T, 0, 0, 0',
	X =  218.594  mm,	Y =   -469.321  mm,	Z =   -340.561  mm,
	W =  90.000 deg,	P =   0.000 deg,	R =   90.000 deg
};
P[195]{
   GP1:
	UF : 0, UT : 6,		CONFIG : 'N U T, 0, 0, 0',
	X =  287.454  mm,	Y =   -430.013  mm,	Z =   -331.997  mm,
	W =  90.000 deg,	P =   0.000 deg,	R =   90.000 deg
};
P[196]{
   GP1:
	UF : 0, UT : 6,		CONFIG : 'N U T, 0, 0, 0',
	X =  305.966  mm,	Y =   -420.083  mm,	Z =   -329.001  mm,
	W =  90.000 deg,	P =   0.000 deg,	R =   90.000 deg
};
P[197]{
   GP1:
	UF : 0, UT : 6,		CONFIG : 'N U T, 0, 0, 0',
	X =  201.102  mm,	Y =   -480.515  mm,	Z =   -330.136  mm,
	W =  90.000 deg,	P =   0.000 deg,	R =   90.000 deg
};
P[198]{
   GP1:
	UF : 0, UT : 6,		CONFIG : 'N U T, 0, 0, 0',
	X =  172.477  mm,	Y =   -500.311  mm,	Z =   -332.957  mm,
	W =  90.000 deg,	P =   0.000 deg,	R =   90.000 deg
};
P[199]{
   GP1:
	UF : 0, UT : 6,		CONFIG : 'N U T, 0, 0, 0',
	X =  185.596  mm,	Y =   -493.154  mm,	Z =   -344.563  mm,
	W =  90.000 deg,	P =   0.000 deg,	R =   90.000 deg
};
P[200]{
   GP1:
	UF : 0, UT : 6,		CONFIG : 'N U T, 0, 0, 0',
	X =  237.683  mm,	Y =   -463.424  mm,	Z =   -340.200  mm,
	W =  90.000 deg,	P =   0.000 deg,	R =   90.000 deg
};
P[201]{
   GP1:
	UF : 0, UT : 6,		CONFIG : 'N U T, 0, 0, 0',
	X =  254.924  mm,	Y =   -452.971  mm,	Z =   -339.103  mm,
	W =  90.000 deg,	P =   0.000 deg,	R =   90.000 deg
};
P[202]{
   GP1:
	UF : 0, UT : 6,		CONFIG : 'N U T, 0, 0, 0',
	X =  271.151  mm,	Y =   -443.214  mm,	Z =   -330.502  mm,
	W =  90.000 deg,	P =   0.000 deg,	R =   90.000 deg
};
P[203]{
   GP1:
	UF : 0, UT : 6,		CONFIG : 'N U T, 0, 0, 0',
	X =  337.121  mm,	Y =   -405.419  mm,	Z =   -329.000  mm,
	W =  90.000 deg,	P =   0.000 deg,	R =   90.000 deg
};
P[204]{
   GP1:
	UF : 0, UT : 6,		CONFIG : 'N U T, 0, 0, 0',
	X =  324.257  mm,	Y =   -413.926  mm,	Z =   -344.965  mm,
	W =  90.000 deg,	P =   0.000 deg,	R =   90.000 deg
};
P[205]{
   GP1:
	UF : 0, UT : 6,		CONFIG : 'N U T, 0, 0, 0',
	X =  221.718  mm,	Y =   -476.870  mm,	Z =   -331.754  mm,
	W =  90.000 deg,	P =   0.000 deg,	R =   90.000 deg
};
P[206]{
   GP1:
	UF : 0, UT : 6,		CONFIG : 'N U T, 0, 0, 0',
	X =  292.570  mm,	Y =   -436.361  mm,	Z =   -329.000  mm,
	W =  90.000 deg,	P =   0.000 deg,	R =   90.000 deg
};
P[207]{
   GP1:
	UF : 0, UT : 6,		CONFIG : 'N U T, 0, 0, 0',
	X =  308.415  mm,	Y =   -427.634  mm,	Z =   -331.779  mm,
	W =  90.000 deg,	P =   0.000 deg,	R =   90.000 deg
};
P[208]{
   GP1:
	UF : 0, UT : 6,		CONFIG : 'N U T, 0, 0, 0',
	X =  206.369  mm,	Y =   -486.847  mm,	Z =   -329.000  mm,
	W =  90.000 deg,	P =   0.000 deg,	R =   90.000 deg
};
P[209]{
   GP1:
	UF : 0, UT : 6,		CONFIG : 'N U T, 0, 0, 0',
	X =  192.757  mm,	Y =   -497.007  mm,	Z =   -342.135  mm,
	W =  90.000 deg,	P =   0.000 deg,	R =   90.000 deg
};
P[210]{
   GP1:
	UF : 0, UT : 6,		CONFIG : 'N U T, 0, 0, 0',
	X =  235.408  mm,	Y =   -472.525  mm,	Z =   -340.269  mm,
	W =  90.000 deg,	P =   0.000 deg,	R =   90.000 deg
};
P[211]{
   GP1:
	UF : 0, UT : 6,		CONFIG : 'N U T, 0, 0, 0',
	X =  277.326  mm,	Y =   -447.892  mm,	Z =   -329.042  mm,
	W =  90.000 deg,	P =   0.000 deg,	R =   90.000 deg
};
P[212]{
   GP1:
	UF : 0, UT : 6,		CONFIG : 'N U T, 0, 0, 0',
	X =  321.012  mm,	Y =   -424.478  mm,	Z =   -341.674  mm,
	W =  90.000 deg,	P =   0.000 deg,	R =   90.000 deg
};
P[213]{
   GP1:
	UF : 0, UT : 6,		CONFIG : 'N U T, 0, 0, 0',
	X =  325.701  mm,	Y =   -430.727  mm,	Z =   -329.068  mm,
	W =  90.000 deg,	P =   0.000 deg,	R =   90.000 deg
};
P[214]{
   GP1:
	UF : 0, UT : 6,		CONFIG : 'N U T, 0, 0, 0',
	X =  241.616  mm,	Y =   -480.522  mm,	Z =   -329.106  mm,
	W =  90.000 deg,	P =   0.000 deg,	R =   90.000 deg
};
P[215]{
   GP1:
	UF : 0, UT : 6,		CONFIG : 'N U T, 0, 0, 0',
	X =  197.508  mm,	Y =   -506.852  mm,	Z =   -344.034  mm,
	W =  90.000 deg,	P =   0.000 deg,	R =   90.000 deg
};
P[216]{
   GP1:
	UF : 0, UT : 6,		CONFIG : 'N U T, 0, 0, 0',
	X =  281.959  mm,	Y =   -458.358  mm,	Z =   -331.964  mm,
	W =  90.000 deg,	P =   0.000 deg,	R =   90.000 deg
};
P[217]{
   GP1:
	UF : 0, UT : 6,		CONFIG : 'N U T, 0, 0, 0',
	X =  347.298  mm,	Y =   -422.588  mm,	Z =   -330.516  mm,
	W =  90.000 deg,	P =   0.000 deg,	R =   90.000 deg
};
P[218]{
   GP1:
	UF : 0, UT : 6,		CONFIG : 'N U T, 0, 0, 0',
	X =  334.562  mm,	Y =   -430.572  mm,	Z =   -331.605  mm,
	W =  90.000 deg,	P =   0.000 deg,	R =   90.000 deg
};
P[219]{
   GP1:
	UF : 0, UT : 6,		CONFIG : 'N U T, 0, 0, 0',
	X =  316.746  mm,	Y =   -440.509  mm,	Z =   -330.565  mm,
	W =  90.000 deg,	P =   0.000 deg,	R =   90.000 deg
};
P[220]{
   GP1:
	UF : 0, UT : 6,		CONFIG : 'N U T, 0, 0, 0',
	X =  264.740  mm,	Y =   -470.189  mm,	Z =   -329.022  mm,
	W =  90.000 deg,	P =   0.000 deg,	R =   90.000 deg
};
P[221]{
   GP1:
	UF : 0, UT : 6,		CONFIG : 'N U T, 0, 0, 0',
	X =  213.382  mm,	Y =   -500.167  mm,	Z =   -329.067  mm,
	W =  90.000 deg,	P =   0.000 deg,	R =   90.000 deg
};
P[222]{
   GP1:
	UF : 0, UT : 6,		CONFIG : 'N U T, 0, 0, 0',
	X =  182.650  mm,	Y =   -517.700  mm,	Z =   -329.000  mm,
	W =  90.000 deg,	P =   0.000 deg,	R =   90.000 deg
};
P[223]{
   GP1:
	UF : 0, UT : 6,		CONFIG : 'N U T, 0, 0, 0',
	X =  230.636  mm,	Y =   -490.762  mm,	Z =   -329.039  mm,
	W =  90.000 deg,	P =   0.000 deg,	R =   90.000 deg
};
P[224]{
   GP1:
	UF : 0, UT : 6,		CONFIG : 'N U T, 0, 0, 0',
	X =  299.932  mm,	Y =   -450.773  mm,	Z =   -331.827  mm,
	W =  90.000 deg,	P =   0.000 deg,	R =   90.000 deg
};
P[225]{
   GP1:
	UF : 0, UT : 6,		CONFIG : 'N U T, 0, 0, 0',
	X =  249.896  mm,	Y =   -480.755  mm,	Z =   -329.002  mm,
	W =  90.000 deg,	P =   0.000 deg,	R =   90.000 deg
};
P[226]{
   GP1:
	UF : 0, UT : 6,		CONFIG : 'N U T, 0, 0, 0',
	X =  195.088  mm,	Y =   -512.788  mm,	Z =   -330.121  mm,
	W =  90.000 deg,	P =   0.000 deg,	R =   90.000 deg
};
P[227]{
   GP1:
	UF : 0, UT : 6,		CONFIG : 'N U T, 0, 0, 0',
	X =  280.354  mm,	Y =   -464.983  mm,	Z =   -329.029  mm,
	W =  90.000 deg,	P =   0.000 deg,	R =   90.000 deg
};
P[228]{
   GP1:
	UF : 0, UT : 6,		CONFIG : 'N U T, 0, 0, 0',
	X =  326.977  mm,	Y =   -443.919  mm,	Z =   -330.464  mm,
	W =  90.000 deg,	P =   0.000 deg,	R =   90.000 deg
};
P[229]{
   GP1:
	UF : 0, UT : 6,		CONFIG : 'N U T, 0, 0, 0',
	X =  212.811  mm,	Y =   -510.913  mm,	Z =   -330.006  mm,
	W =  90.000 deg,	P =   0.000 deg,	R =   90.000 deg
};
P[230]{
   GP1:
	UF : 0, UT : 6,		CONFIG : 'N U T, 0, 0, 0',
	X =  242.213  mm,	Y =   -494.095  mm,	Z =   -342.776  mm,
	W =  90.000 deg,	P =   0.000 deg,	R =   90.000 deg
};
P[231]{
   GP1:
	UF : 0, UT : 6,		CONFIG : 'N U T, 0, 0, 0',
	X =  298.403  mm,	Y =   -461.781  mm,	Z =   -329.019  mm,
	W =  90.000 deg,	P =   0.000 deg,	R =   90.000 deg
};
P[232]{
   GP1:
	UF : 0, UT : 6,		CONFIG : 'N U T, 0, 0, 0',
	X =  225.694  mm,	Y =   -505.041  mm,	Z =   -329.013  mm,
	W =  90.000 deg,	P =   0.000 deg,	R =   90.000 deg
};
P[233]{
   GP1:
	UF : 0, UT : 6,		CONFIG : 'N U T, 0, 0, 0',
	X =  231.971  mm,	Y =   -501.687  mm,	Z =   -329.039  mm,
	W =  90.000 deg,	P =   0.000 deg,	R =   90.000 deg
};
P[234]{
   GP1:
	UF : 0, UT : 6,		CONFIG : 'N U T, 0, 0, 0',
	X =  310.353  mm,	Y =   -456.395  mm,	Z =   -329.008  mm,
	W =  90.000 deg,	P =   0.000 deg,	R =   90.000 deg
};
P[235]{
   GP1:
	UF : 0, UT : 6,		CONFIG : 'N U T, 0, 0, 0',
	X =  316.421  mm,	Y =   -452.825  mm,	Z =   -329.000  mm,
	W =  90.000 deg,	P =   0.000 deg,	R =   90.000 deg
};
P[236]{
   GP1:
	UF : 0, UT : 6,		CONFIG : 'N U T, 0, 0, 0',
	X =  308.920  mm,	Y =   -465.983  mm,	Z =   -329.008  mm,
	W =  90.000 deg,	P =   0.000 deg,	R =   90.000 deg
};
P[237]{
   GP1:
	UF : 0, UT : 6,		CONFIG : 'N U T, 0, 0, 0',
	X =  239.601  mm,	Y =   -506.070  mm,	Z =   -329.069  mm,
	W =  90.000 deg,	P =   0.000 deg,	R =   90.000 deg
};
P[238]{
   GP1:
	UF : 0, UT : 6,		CONFIG : 'N U T, 0, 0, 0',
	X =  222.365  mm,	Y =   -515.873  mm,	Z =   -329.000  mm,
	W =  90.000 deg,	P =   0.000 deg,	R =   90.000 deg
};
P[239]{
   GP1:
	UF : 0, UT : 6,		CONFIG : 'N U T, 0, 0, 0',
	X =  325.840  mm,	Y =   -456.566  mm,	Z =   -342.918  mm,
	W =  90.000 deg,	P =   0.000 deg,	R =   90.000 deg
};
P[240]{
   GP1:
	UF : 0, UT : 6,		CONFIG : 'N U T, 0, 0, 0',
	X =  357.338  mm,	Y =   -439.893  mm,	Z =   -329.000  mm,
	W =  90.000 deg,	P =   0.000 deg,	R =   90.000 deg
};
P[241]{
   GP1:
	UF : 0, UT : 6,		CONFIG : 'N U T, 0, 0, 0',
	X =  344.350  mm,	Y =   -447.657  mm,	Z =   -330.589  mm,
	W =  90.000 deg,	P =   0.000 deg,	R =   90.000 deg
};
P[242]{
   GP1:
	UF : 0, UT : 6,		CONFIG : 'N U T, 0, 0, 0',
	X =  292.438  mm,	Y =   -477.174  mm,	Z =   -331.946  mm,
	W =  90.000 deg,	P =   0.000 deg,	R =   90.000 deg
};
P[243]{
   GP1:
	UF : 0, UT : 6,		CONFIG : 'N U T, 0, 0, 0',
	X =  274.843  mm,	Y =   -487.492  mm,	Z =   -329.012  mm,
	W =  90.000 deg,	P =   0.000 deg,	R =   90.000 deg
};
P[244]{
   GP1:
	UF : 0, UT : 6,		CONFIG : 'N U T, 0, 0, 0',
	X =  257.698  mm,	Y =   -497.487  mm,	Z =   -329.013  mm,
	W =  90.000 deg,	P =   0.000 deg,	R =   90.000 deg
};
P[245]{
   GP1:
	UF : 0, UT : 6,		CONFIG : 'N U T, 0, 0, 0',
	X =  205.679  mm,	Y =   -527.553  mm,	Z =   -344.515  mm,
	W =  90.000 deg,	P =   0.000 deg,	R =   90.000 deg
};
P[246]{
   GP1:
	UF : 0, UT : 6,		CONFIG : 'N U T, 0, 0, 0',
	X =  192.735  mm,	Y =   -535.298  mm,	Z =   -329.042  mm,
	W =  90.000 deg,	P =   0.000 deg,	R =   90.000 deg
};
P[247]{
   GP1:
	UF : 0, UT : 6,		CONFIG : 'N U T, 0, 0, 0',
	X =  199.890  mm,	Y =   -548.244  mm,	Z =   -329.000  mm,
	W =  90.000 deg,	P =   0.000 deg,	R =   90.000 deg
};
P[248]{
   GP1:
	UF : 0, UT : 6,		CONFIG : 'N U T, 0, 0, 0',
	X =  213.173  mm,	Y =   -540.691  mm,	Z =   -330.250  mm,
	W =  90.000 deg,	P =   0.000 deg,	R =   90.000 deg
};
P[249]{
   GP1:
	UF : 0, UT : 6,		CONFIG : 'N U T, 0, 0, 0',
	X =  230.358  mm,	Y =   -530.659  mm,	Z =   -329.989  mm,
	W =  90.000 deg,	P =   0.000 deg,	R =   90.000 deg
};
P[250]{
   GP1:
	UF : 0, UT : 6,		CONFIG : 'N U T, 0, 0, 0',
	X =  247.811  mm,	Y =   -520.778  mm,	Z =   -329.000  mm,
	W =  90.000 deg,	P =   0.000 deg,	R =   90.000 deg
};
P[251]{
   GP1:
	UF : 0, UT : 6,		CONFIG : 'N U T, 0, 0, 0',
	X =  265.508  mm,	Y =   -510.586  mm,	Z =   -329.000  mm,
	W =  90.000 deg,	P =   0.000 deg,	R =   90.000 deg
};
P[252]{
   GP1:
	UF : 0, UT : 6,		CONFIG : 'N U T, 0, 0, 0',
	X =  282.543  mm,	Y =   -500.692  mm,	Z =   -329.000  mm,
	W =  90.000 deg,	P =   0.000 deg,	R =   90.000 deg
};
P[253]{
   GP1:
	UF : 0, UT : 6,		CONFIG : 'N U T, 0, 0, 0',
	X =  299.785  mm,	Y =   -490.752  mm,	Z =   -331.587  mm,
	W =  90.000 deg,	P =   0.000 deg,	R =   90.000 deg
};
P[254]{
   GP1:
	UF : 0, UT : 6,		CONFIG : 'N U T, 0, 0, 0',
	X =  317.146  mm,	Y =   -480.700  mm,	Z =   -339.097  mm,
	W =  90.000 deg,	P =   0.000 deg,	R =   90.000 deg
};
P[255]{
   GP1:
	UF : 0, UT : 6,		CONFIG : 'N U T, 0, 0, 0',
	X =  334.570  mm,	Y =   -470.575  mm,	Z =   -331.336  mm,
	W =  90.000 deg,	P =   0.000 deg,	R =   90.000 deg
};
P[256]{
   GP1:
	UF : 0, UT : 6,		CONFIG : 'N U T, 0, 0, 0',
	X =  351.785  mm,	Y =   -460.601  mm,	Z =   -330.492  mm,
	W =  90.000 deg,	P =   0.000 deg,	R =   90.000 deg
};
P[257]{
   GP1:
	UF : 0, UT : 6,		CONFIG : 'N U T, 0, 0, 0',
	X =  364.957  mm,	Y =   -453.093  mm,	Z =   -342.229  mm,
	W =  90.000 deg,	P =   0.000 deg,	R =   90.000 deg
};
P[258]{
   GP1:
	UF : 0, UT : 6,		CONFIG : 'N U T, 0, 0, 0',
	X =  210.000  mm,	Y =   -375.000  mm,	Z =   -250.000  mm,
	W =  90.000 deg,	P =   0.000 deg,	R =   90.000 deg
};
/END
